# EPICS alarm handler configuration: alh_files/mgnt_dmp.alhConfig
GROUP NULL MGNT:DMP1:1
   $COMMAND edm -x -eolc -noedit mgnt_dmp1_main.edl

$ALIAS DMP1
$GUIDANCE
dump Magnet
   Group Name: MGNT:DMP1:1
   Summary PV:  MGNT:DMP1:1:STATSUMY
$END

   INCLUDE MGNT:DMP1:1 ./mgnt_dmp1_bend.alhConfig
   INCLUDE MGNT:DMP1:1 ./mgnt_dmp1_lgps.alhConfig
   INCLUDE MGNT:DMP1:1 ./mgnt_dmp1_quad.alhConfig
   INCLUDE MGNT:DMP1:1 ./mgnt_dmp1_xcor.alhConfig
   INCLUDE MGNT:DMP1:1 ./mgnt_dmp1_ycor.alhConfig
